{attribute 'GeneratedUsingTerminal: KL2521'}
{attribute addProperty BoxType "KL2521"}
{attribute addProperty Id "Channel_1AT %Q*Channel_03CEAA5E0"}
{attribute addProperty CRC "3589488903"}
{attribute addProperty Size "0"}
TYPE KL2521_D5F34107 :
STRUCT
	{attribute addProperty Name "Channel_1"}
	Channel_1 : Channel_03CEAA5E;
END_STRUCT
END_TYPE

(* stored: Version 1.2.0.0, ProductVersion 3.1.4024.9
   DUT KL2521_D5F34107: Id {8d142029-b1cf-427f-8e2c-f626e755452b} *)
